(* IEC 61131-3 sources: AXOpen/src/components.keyence.vision/ctrl/src/Axo_IV3 (part 4) *)

            _programNumber := inProgramNumber;
            ChangeProgram := ChangeProgramTask.Invoke(THIS);
        END_METHOD

        METHOD PROTECTED OVERRIDE ManualControl
            THIS._isManuallyControllable := true;
            _programNumber := RequiredProgramNumber;
        END_METHOD

        ///<summary>
        /// Restores this component into intial state.
        ///</summary>
        METHOD PUBLIC OVERRIDE Restore
            VAR
                _index : INT;
            END_VAR
            Status.Action.Id := UINT#0;
            Status.Error.Id  := UINT#0;

            _progress       :=   INT#0;
            _retVal    :=   WORD#0;

            Outputs.CommandControl.TriggerRequest                               := FALSE;
            Outputs.CommandControl.MasterRegistrationRequest                    := FALSE;
            Outputs.CommandControl.ProgramSwitchingRequest                      := FALSE;
            Outputs.CommandControl.WarningClearRequest                          := FALSE;
            Outputs.CommandControl.StatisticsResetRequest                       := FALSE;
            Outputs.CommandControl.BufferClearRequest                           := FALSE;
            Outputs.CommandControl.SdCardSavingStopRequest                      := FALSE;
            Outputs.CommandControl.SettingValueChangeRequest                    := FALSE;
            Outputs.CommandControl.ResultAcquisitionCompleteNotification        := FALSE;
            Outputs.CommandControl.ProgramNo                                    := UINT#0;
            Outputs.CommandControl.Function_1                                   := WORD#0;
            Outputs.CommandControl.Function_2                                   := DWORD#0;

            FOR _index := 0 TO 11 DO
                _data_in[_index] := BYTE#0;
                _data_out_12[_index] := BYTE#0;
            END_FOR;

            FOR _index := 12 TO 27 DO
                _data_in[_index] := BYTE#0;
            END_FOR;

            _word           :=   WORD#0;
            _dword          :=   DWORD#0;

            TriggerTask.Restore();
            ChangeProgramTask.Restore();
            HardwareDiagnosticsTask.Restore();

            Status.Action.Id := UINT#50;
            RestoreTask.DoneWhen(TRUE);

        END_METHOD

        METHOD PRIVATE CallTimers
            VAR_INPUT
                signal : BOOL;
            END_VAR

            _infoTimer.OnDelay(THIS, signal AND Config.InfoTime > T#0S ,Config.InfoTime);
            _errorTimer.OnDelay(THIS, signal AND Config.ErrorTime > T#0S , Config.ErrorTime);

        END_METHOD

    END_CLASS
END_NAMESPACE
